(* IEC 61131-3 sources: AXOpen/src/data/ctrl/test, 10 files *)

(* ---- AxoDataCrudTask.st ---- *)
USING AXOpen.Core;
USING AXOpen.Rtc;
USING AxUnit;

NAMESPACE DummyNmspc
        {TestFixture}
        {S7.extern=ReadWrite}
        CLASS DummyClass

            {Test}
            METHOD PUBLIC Create_sets_identifier
                AxUnit.Assert.Equal(TRUE, TRUE);
            END_METHOD

        END_CLASS
END_NAMESPACE

(* ---- AxoDataCrudTaskEntityExistsSatisfiedTests.st ---- *)
USING AXOpen.Core;
USING AXOpen.Data;
USING AxUnit;

NAMESPACE AXOpen.Data
    {TestFixture}
    {S7.extern=ReadWrite}
    CLASS AxoDataCrudTaskEntityExistsSatisfiedTests
        VAR
            _state : AxoDataCrudTaskEntityExistsSatisfied;
        END_VAR

        {Test}
        METHOD PUBLIC Satisfy_sets_status_and_exist_flag
            VAR
                existsAfterFirstRead : BOOL;
                existsAfterSecondRead : BOOL;
            END_VAR

            _state.Satisfy(eAxoTaskState#Done, TRUE);
            existsAfterFirstRead := _state.Exist();
            existsAfterSecondRead := _state.Exist();

            AxUnit.Assert.Equal(eAxoTaskState#Done, _state.Status);
            AxUnit.Assert.Equal(TRUE, existsAfterFirstRead);
            AxUnit.Assert.Equal(FALSE, existsAfterSecondRead);
        END_METHOD

        {Test}
        METHOD PUBLIC Satisfy_with_false_clears_exist_flag
            VAR
                existsAfterRead : BOOL;
            END_VAR

            _state.Satisfy(eAxoTaskState#Busy, FALSE);
            existsAfterRead := _state.Exist();

            AxUnit.Assert.Equal(eAxoTaskState#Busy, _state.Status);
            AxUnit.Assert.Equal(FALSE, existsAfterRead);
            AxUnit.Assert.Equal(FALSE, _state.Exist());
        END_METHOD
    END_CLASS
END_NAMESPACE

(* ---- AxoDataExchangeTaskTests.st ---- *)
USING AXOpen.Core;
USING AXOpen.Rtc;
USING AxUnit;

NAMESPACE AXOpen.Data
    NAMESPACE AxoDataExchangeTaskTests
        {S7.extern=ReadWrite}
        CLASS TestContext IMPLEMENTS IAxoContext
            VAR PROTECTED
                _openCounter : ULINT;
                _closeCounter : ULINT;
                _identityCounter : ULINT;
             END_VAR
            METHOD PUBLIC Open : ULINT
                _openCounter := _openCounter + ULINT#1;
            END_METHOD

            METHOD PUBLIC Close : ULINT
                _closeCounter := _closeCounter + ULINT#1;
            END_METHOD

            METHOD PUBLIC OpenCycleCount : ULINT
                OpenCycleCount := _openCounter;
            END_METHOD

            METHOD PUBLIC ClosedCycleCount : ULINT
                ClosedCycleCount := _closeCounter;
            END_METHOD

            METHOD PUBLIC CreateIdentity : ULINT
                _identityCounter := _identityCounter + ULINT#1;
                CreateIdentity := _identityCounter;
            END_METHOD

            METHOD PUBLIC GetRtc : IAxoRtc ; END_METHOD

            METHOD PUBLIC InjectRtc VAR_INPUT Rtc : IAxoRtc; END_VAR ; END_METHOD

            VAR PRIVATE
                NULL_LOGGER : _NULL_LOGGER;
            END_VAR
            METHOD PUBLIC GetLogger : AXOpen.Logging.IAxoLogger GetLogger := NULL_LOGGER; END_METHOD
            METHOD PUBLIC InjectLogger VAR_INPUT _logger : AXOpen.Logging.IAxoLogger; END_VAR ; END_METHOD
        END_CLASS

        {TestFixture}
        {S7.extern=ReadWrite}
        CLASS AxoDataExchangeTask_Tests
            VAR PROTECTED
                _context : TestContext;
                _dataExchangeTask : AxoDataCrudTask;
            END_VAR

            {Test}
            METHOD PUBLIC InvokeWithIdentifier_sets_identifier
                VAR
                    expected : STRING[254];
                END_VAR
                _dataExchangeTask.Initialize(_context);
                _context.Open();
                expected := 'CreateRecordIdentifier';
                _dataExchangeTask.Invoke(expected);
                _context.Close();
                AxUnit.Assert.Equal(TRUE, _dataExchangeTask.DataEntityIdentifier = expected);
            END_METHOD

        END_CLASS
    END_NAMESPACE
END_NAMESPACE

(* ---- AxoDataExchangeTests.st ---- *)
USING AXOpen.Core;
USING AXOpen.Rtc;
USING AxUnit;

NAMESPACE AXOpen.Data
    NAMESPACE AxoDataExchangeTests
        CLASS TestContext IMPLEMENTS IAxoContext
            VAR PROTECTED
                _openCounter : ULINT;
                _closeCounter : ULINT;
                _identityCounter : ULINT;
             END_VAR
            METHOD PUBLIC Open : ULINT
                _openCounter := _openCounter + ULINT#1;
            END_METHOD

            METHOD PUBLIC Close : ULINT
                _closeCounter := _closeCounter + ULINT#1;
            END_METHOD

            METHOD PUBLIC OpenCycleCount : ULINT
                OpenCycleCount := _openCounter;
            END_METHOD

            METHOD PUBLIC ClosedCycleCount : ULINT
                ClosedCycleCount := _closeCounter;
            END_METHOD

            METHOD PUBLIC CreateIdentity : ULINT
                _identityCounter := _identityCounter + ULINT#1;
                CreateIdentity := _identityCounter;
            END_METHOD

            METHOD PUBLIC GetRtc : IAxoRtc ; END_METHOD

            METHOD PUBLIC InjectRtc VAR_INPUT Rtc : IAxoRtc; END_VAR ; END_METHOD
            VAR PRIVATE
                NULL_LOGGER : _NULL_LOGGER;
            END_VAR
            METHOD PUBLIC GetLogger : AXOpen.Logging.IAxoLogger GetLogger := NULL_LOGGER; END_METHOD
            METHOD PUBLIC InjectLogger VAR_INPUT _logger : AXOpen.Logging.IAxoLogger; END_VAR ; END_METHOD
        END_CLASS

        {TestFixture}
        CLASS AxoDataExchange_Tests
            VAR PROTECTED
                _context : TestContext;
                _dataExchange : AxoDataExchange;
            END_VAR

            {Test}
            METHOD PUBLIC Create_sets_identifier
                VAR
                    expected : STRING[254];
                END_VAR
                _dataExchange.Initialize(_context);
                _context.Open();
                expected := 'CreateRecordIdentifier';
                _dataExchange.Create(expected);
                _context.Close();
                AxUnit.Assert.Equal(_dataExchange.Operation.DataEntityIdentifier, expected);
            END_METHOD

            {Test}
            METHOD PUBLIC Read_sets_identifier
                VAR
                    expected : STRING[254];
                END_VAR
                _dataExchange.Initialize(_context);
                _context.Open();
                expected := 'ReadRecordIdentifier';
                _dataExchange.Read(expected);
                _context.Close();
                AxUnit.Assert.Equal(_dataExchange.Operation.DataEntityIdentifier, expected);
            END_METHOD

            {Test}
            METHOD PUBLIC Update_sets_identifier
                VAR
                    expected : STRING[254];
                END_VAR
                _dataExchange.Initialize(_context);
                _context.Open();
                expected := 'UpdateRecordIdentifier';
                _dataExchange.Update(expected);
                _context.Close();
                AxUnit.Assert.Equal(_dataExchange.Operation.DataEntityIdentifier, expected);
            END_METHOD

            {Test}
            METHOD PUBLIC Delete_sets_identifier
                VAR
                    expected : STRING[254];
                END_VAR
                _dataExchange.Initialize(_context);
                _context.Open();
                expected := 'DeleteRecordIdentifier';
                _dataExchange.Delete(expected);
                _context.Close();
                AxUnit.Assert.Equal(_dataExchange.Operation.DataEntityIdentifier, expected);
            END_METHOD

            {Test}
            METHOD PUBLIC EntityExist_sets_identifier
                VAR
                    expected : STRING[254];
                END_VAR
                _dataExchange.Initialize(_context);
                _context.Open();
                expected := 'EntityExistRecordIdentifier';
                _dataExchange.EntityExist(expected);
                _context.Close();
                AxUnit.Assert.Equal(_dataExchange.Operation.DataEntityIdentifier, expected);
            END_METHOD

            {Test}
            METHOD PUBLIC CreateOrUpdate_sets_identifier
                VAR
                    expected : STRING[254];
                END_VAR
                _dataExchange.Initialize(_context);
                _context.Open();
                expected := 'CreateOrUpdateRecordIdentifier';
                _dataExchange.CreateOrUpdate(expected);
                _context.Close();
                AxUnit.Assert.Equal(_dataExchange.Operation.DataEntityIdentifier, expected);
            END_METHOD
        END_CLASS
    END_NAMESPACE
END_NAMESPACE

(* ---- AxoDataLocalExchangeTest.st ---- *)
USING AXOpen.Messaging.Static;
USING AXOpen.Core;
USING AXOpen.Core.Dummies;
USING AXOpen.Data;

NAMESPACE AXOpen.Data
    CLASS _DataStorage_template EXTENDS AxoDataLocalExchange
        VAR CONSTANT
            LOWBOUND : DINT := 0;
            HIGHBOUND : DINT := 10;
        END_VAR
        VAR PUBLIC
            Payload : _EntityTemplate_;
            Storage : ARRAY[LOWBOUND..HIGHBOUND] OF _EntityTemplate_;
        END_VAR

        METHOD PUBLIC OVERRIDE Create : IAxoTaskState
            VAR_INPUT
                inIdentifier : STRING[254];
            END_VAR
            VAR
                tmpSlot : DINT;
             END_VAR

            dataExchangeTask.Status := eAxoTaskState#Busy;
            operation := eCrudOperation#Create;

            tmpSlot :=THIS.GetFreeSlot();
            IF(tmpSlot >= 0) THEN
                Payload.DataEntityId :=  inIdentifier;
                Storage[tmpSlot] :=  Payload;
                dataExchangeTask.Status := eAxoTaskState#Done;
            ELSE
                dataExchangeTask.Status := eAxoTaskState#Error;
            END_IF;

            Create := dataExchangeTask;
        END_METHOD

        METHOD PUBLIC OVERRIDE Read : IAxoTaskState
            VAR_INPUT
                inIdentifier : STRING[254];
            END_VAR
            VAR
                tmpStorage : REF_TO ARRAY[*] OF IAxoDataEntity;
                tmpEntity : IAxoDataEntity;
                tmpSlot : DINT;
             END_VAR

            dataExchangeTask.Status := eAxoTaskState#Busy;
            operation := eCrudOperation#Read;
            tmpSlot := THIS.LocateSlot(inIdentifier);
            IF(tmpSlot >= LOWBOUND && tmpSlot <= HIGHBOUND) THEN
                Payload := Storage[tmpSlot];
                dataExchangeTask.Status := eAxoTaskState#Done;
            ELSE
                dataExchangeTask.Status := eAxoTaskState#Error;
            END_IF;

            Read := dataExchangeTask;
        END_METHOD

        METHOD PUBLIC OVERRIDE Update : IAxoTaskState
            VAR_INPUT
                inIdentifier : STRING[254];
            END_VAR
            VAR
                tmpSlot : DINT;
            END_VAR
            dataExchangeTask.Status := eAxoTaskState#Busy;
            operation := eCrudOperation#Update;

            tmpSlot := THIS.LocateSlot(inIdentifier);
            IF(tmpSlot >= LOWBOUND && tmpSlot <= HIGHBOUND) THEN
                Payload := Storage[tmpSlot];
                dataExchangeTask.Status := eAxoTaskState#Done;
            ELSE
                dataExchangeTask.Status := eAxoTaskState#Error;
            END_IF;

            Update := dataExchangeTask;
        END_METHOD

        METHOD PUBLIC OVERRIDE Delete : IAxoTaskState
            VAR_INPUT
                inIdentifier : STRING[254];
            END_VAR

            dataExchangeTask.Status := eAxoTaskState#Busy;
            operation := eCrudOperation#Delete;

            Storage[THIS.LocateSlot(inIdentifier)].DataEntityId := '';
            dataExchangeTask.Status := eAxoTaskState#Done;
            Delete := dataExchangeTask;
        END_METHOD

        METHOD PUBLIC OVERRIDE EntityExist : IAxoDataCrudTaskEntityExistState
            VAR_INPUT
                inIdentifier : STRING[254];
            END_VAR
            ;
        END_METHOD

        METHOD PUBLIC OVERRIDE CreateOrUpdate : IAxoTaskState
            VAR_INPUT
                inIdentifier : STRING[254];
            END_VAR
            dataExchangeTask.Status := eAxoTaskState#Done;
            CreateOrUpdate := dataExchangeTask;
        END_METHOD

        METHOD PUBLIC OVERRIDE Restore
            ;
        END_METHOD

        METHOD PRIVATE GetFreeSlot : DINT
            VAR
                i : DINT;
                s : IAxoDataEntity;
            END_VAR
            GetFreeSlot := -1;
            FOR i := LOWBOUND TO HIGHBOUND DO
                IF(Storage[i].DataEntityId = '') THEN
                     GetFreeSlot := i;
                     RETURN;
                END_IF;
            END_FOR;
        END_METHOD

        METHOD PRIVATE LocateSlot : DINT
            VAR_INPUT
                inIdentifier : STRING[254];
            END_VAR
            VAR
                i : DINT;
                s : IAxoDataEntity;
            END_VAR
            LocateSlot := -1;
            FOR i := LOWBOUND TO HIGHBOUND DO
                IF(Storage[i].DataEntityId = inIdentifier) THEN
                    LocateSlot := i;
                     RETURN;
                END_IF;
            END_FOR;
        END_METHOD
    END_CLASS

    {TestFixture}
    {S7.extern=ReadWrite}
    CLASS AxoDataLocalExchangeTests
        VAR
            context : Context;
            rootObject : MockAxoObject;
            storageController : _DataStorage_template;
            s : ARRAY[0..10] OF _EntityTemplate_;
            rtm : MockAxoRtm;
            rtc : MockAxoRtc;
        END_VAR

        {FixtureSetup}
        METHOD PUBLIC TestFixtureSetup
            VAR
                index : INT;
            END_VAR
            context.InitializeRootObject(rootObject);
            context.InjectRtc(rtc);
            context.InjectRtm(rtm);
        END_METHOD

        {Test}
        METHOD PUBLIC create_new_entity_with_identifier
            VAR
                index : INT;
            END_VAR

            storageController.Payload.DataEntityId := 'NON-ID';
            storageController.Payload._hello := 'HEY';
            storageController.Payload._someNumber := 1;
            storageController.Create('ID');

            storageController.Payload.DataEntityId := 'NON-ID';
            storageController.Payload._hello := 'HEY-2';
            storageController.Payload._someNumber := 2;
            storageController.Create('ID-2');

            storageController.Read('ID');

            AxUnit.Assert.Equal(storageController.Payload._hello = 'HEY' , TRUE);
            AxUnit.Assert.Equal(storageController.Payload.DataEntityId = 'ID' , TRUE);
            AxUnit.Assert.Equal(storageController.Payload._someNumber , 1);
        END_METHOD

        {Test}
        METHOD PUBLIC read_new_entity_with_identifier
            VAR
                index : INT;
            END_VAR

            storageController.Payload.DataEntityId := 'NON-ID';
            storageController.Payload._hello := 'HEY';
            storageController.Payload._someNumber := 1;
            storageController.Create('ID');

            storageController.Payload.DataEntityId := 'NON-ID';
            storageController.Payload._hello := 'TO_BE_READ';
            storageController.Payload._someNumber := 2;
            storageController.Create('READ-ID');

            storageController.Read('READ-ID');

            AxUnit.Assert.Equal(storageController.Payload._hello = 'TO_BE_READ' , TRUE);
            AxUnit.Assert.Equal(storageController.Payload.DataEntityId = 'READ-ID' , TRUE);
            AxUnit.Assert.Equal(storageController.Payload._someNumber , 2);
        END_METHOD

        {Test}
        METHOD PUBLIC delet_entity_with_identifier
            VAR
                index : INT;
            END_VAR

            storageController.Payload.DataEntityId := 'NON-ID';
            storageController.Payload._hello := 'HEY';
            storageController.Payload._someNumber := 1;
            storageController.Create('ID');

            storageController.Payload.DataEntityId := 'NON-ID';
            storageController.Payload._hello := 'TO_BE_READ';
            storageController.Payload._someNumber := 2;
            storageController.Create('DELETE-ID');

            storageController.Delete('DELETE-ID');

            storageController.Read('DELETE-ID');

            AxUnit.Assert.Equal( storageController.Read('DELETE-ID').HasError() , TRUE);
        END_METHOD
    END_CLASS

    CLASS _EntityTemplate_ EXTENDS AxoDataEntity
        VAR PUBLIC
            _hello : STRING;
            _someNumber : INT;
        END_VAR
    END_CLASS
    CLASS Context EXTENDS MockAxoContext
        VAR

        END_VAR
        METHOD OVERRIDE Main
            ;
        END_METHOD
    END_CLASS
END_NAMESPACE

(* ---- AxoDataPersistentExchangeTaskTests.st ---- *)
USING AXOpen.Core;
USING AXOpen.Rtc;
USING AxUnit;

NAMESPACE AXOpen.Data
    NAMESPACE AxoDataPersistentExchangeTaskTests
        {S7.extern=ReadWrite}
        CLASS TestContext IMPLEMENTS IAxoContext
            VAR PROTECTED
                _openCounter : ULINT;
                _closeCounter : ULINT;
                _identityCounter : ULINT;
             END_VAR
            METHOD PUBLIC Open : ULINT
                _openCounter := _openCounter + ULINT#1;
            END_METHOD

            METHOD PUBLIC Close : ULINT
                _closeCounter := _closeCounter + ULINT#1;
            END_METHOD

            METHOD PUBLIC OpenCycleCount : ULINT
                OpenCycleCount := _openCounter;
            END_METHOD

            METHOD PUBLIC ClosedCycleCount : ULINT
                ClosedCycleCount := _closeCounter;
            END_METHOD

            METHOD PUBLIC CreateIdentity : ULINT
                _identityCounter := _identityCounter + ULINT#1;
                CreateIdentity := _identityCounter;
            END_METHOD

            METHOD PUBLIC GetRtc : IAxoRtc ; END_METHOD

            METHOD PUBLIC InjectRtc VAR_INPUT Rtc : IAxoRtc; END_VAR ; END_METHOD

            VAR PRIVATE
                NULL_LOGGER : _NULL_LOGGER;
            END_VAR
            METHOD PUBLIC GetLogger : AXOpen.Logging.IAxoLogger GetLogger := NULL_LOGGER; END_METHOD
            METHOD PUBLIC InjectLogger VAR_INPUT _logger : AXOpen.Logging.IAxoLogger; END_VAR ; END_METHOD
        END_CLASS

        {TestFixture}
        {S7.extern=ReadWrite}
        CLASS AxoDataPersistentExchangeTask_Tests
            VAR PROTECTED
                _context : TestContext;
                _dataExchangeTask : AxoDataPersistentCurdTask;
            END_VAR

            {Test}
            METHOD PUBLIC InvokeWithIdentifier_sets_identifier
                VAR
                    expected : STRING[254];
                END_VAR
                _dataExchangeTask.Initialize(_context);
                _context.Open();
                expected := 'UpdateIdentifier';
                _dataExchangeTask.Invoke(expected);
                _context.Close();
                AxUnit.Assert.Equal(TRUE, _dataExchangeTask.DataEntityIdentifier = expected);
            END_METHOD

        END_CLASS
    END_NAMESPACE
END_NAMESPACE

(* ---- AxoDataPersistentExchangeTests.st ---- *)
USING AXOpen.Core;
USING AXOpen.Rtc;
USING AxUnit;

NAMESPACE AXOpen.Data
    NAMESPACE AxoDataPersistentExchangeTests
        {S7.extern=ReadWrite}
        CLASS TestContext EXTENDS Dummies.MockAxoContext
            METHOD PROTECTED OVERRIDE Main
                ;
            END_METHOD
        END_CLASS

        {TestFixture}
        {S7.extern=ReadWrite}
        CLASS AxoDataExchange_Tests
            VAR PROTECTED
                _context : TestContext;
                _rootObject : AxoObject;
                _rtc : AXOpen.Core.Dummies.MockAxoRtc;
                _rtm : AXOpen.Core.Dummies.MockAxoRtm;

                _dataExchange : AxoDataPersistentExchange;

                caller_1 : AxoObject;
                caller_2 : AxoObject;
            END_VAR

            VAR
                _contextBlank : TestContext;
                _dataExchangeBlank : AxoDataPersistentExchange;
                caller_1Blank : AxoObject;
                caller_2Blank : AxoObject;
            END_VAR

            {TestSetup}
            METHOD PUBLIC TestSetup
            // Will be called before MyTest_A AND before Test_B are executed
                _context := _contextBlank;
                _rtm.SetElapsed(LTIME#2s);
                _context.InjectRtm(_rtm);
                _rtc.SetNowUTC(LDATE_AND_TIME#2012-01-12-15:58:12.123);
                _context.InjectRtc(_rtc);
                _context.InitializeRootObject(_rootObject);
                _dataExchange.Run(_rootObject);
                _dataExchange := _dataExchangeBlank;
                caller_1 := caller_1Blank;
                caller_2 := caller_2Blank;
            END_METHOD

            {TestTearDown}
            METHOD PUBLIC TestTearDown
            // Will be called after MyTest_A AND before Test_B where executed
                ;
            END_METHOD

            {FixtureSetup}
            METHOD PUBLIC FixtureSetup
            // Will be called once before the Tests are executed
                ;
            END_METHOD

            {FixtureTearDown}
            METHOD PUBLIC FixtureTearDown
            // Will be called after the Tests where executed
                ;
            END_METHOD

            METHOD PUBLIC RunContextMultipleltipleTimes
                VAR_INPUT
                    cycleCount : INT;
                end_var
                VAR
                    iteration : INT;
                END_VAR
                FOR iteration := 0 TO cycleCount DO
                    _context.Open();
                    _dataExchange.Run(_rootObject);
                    _context.Close();
                END_FOR;
            END_METHOD

            {Test}
            METHOD PUBLIC InvokeRead_NotInvoked_WhenFirstReadDoneNotFinish
                VAR
                    IdentifierCaller_1 : STRING[254];

                    ResultCaller_1 :BOOL;

                    startTime : LDATE_AND_TIME;
                END_VAR
                // initializtion
                startTime := LDATE_AND_TIME#2023-11-11-11:11:11.111;
                _rtc.SetNowUTC(startTime);
                _context.InjectRtc(_rtc);
                caller_1.Run(_rootObject);
                caller_1.Identity :=  _context.CreateIdentity();
                IdentifierCaller_1 := '1';
                _dataExchange.Operation.IsInitialized := true; //simulate intit from .net side

                // needs to simulate + 2 cycles
                THIS.RunContextMultipleltipleTimes(3);

                 //------------------------ INVOKE READ  ------------------------
                _context.Open();
                _dataExchange.Run(_rootObject);

                AxUnit.Assert.Equal(TRUE, _dataExchange.Operation.IsReady());
                ResultCaller_1 := _dataExchange.InvokeRead(caller_1, IdentifierCaller_1);
                AxUnit.Assert.Equal(TRUE, _dataExchange.Operation._EntityId = '');
                AxUnit.Assert.Equal(ResultCaller_1,FALSE);

                _context.Close();

                //------------------------ INVOKE READ  ------------------------
                _context.Open();
                _dataExchange.Run(_rootObject);

                AxUnit.Assert.Equal(TRUE, _dataExchange.Operation.IsReady());
                ResultCaller_1 := _dataExchange.InvokeRead(caller_1, IdentifierCaller_1);
                AxUnit.Assert.Equal(TRUE, _dataExchange.Operation._EntityId = '');
                AxUnit.Assert.Equal(ResultCaller_1,FALSE);

                _context.Close();

                //------------------------ INVOKE READ  ------------------------
                _context.Open();
                _dataExchange.Run(_rootObject);

                AxUnit.Assert.Equal(TRUE, _dataExchange.Operation.IsReady());
                ResultCaller_1 := _dataExchange.InvokeRead(caller_1, IdentifierCaller_1);
                AxUnit.Assert.Equal(TRUE, _dataExchange.Operation._EntityId = '');
                AxUnit.Assert.Equal(ResultCaller_1,FALSE);

                _context.Close();
            END_METHOD

            {Test}
            METHOD PUBLIC InvokeRead_Invoked_WhenFirstReadDoneFinish
                VAR
                    IdentifierCaller_1 : STRING[254];

                    ResultCaller_1 :BOOL;

                    startTime : LDATE_AND_TIME;
                END_VAR
                // initializtion
                startTime := LDATE_AND_TIME#2023-11-11-11:11:11.111;
                _rtc.SetNowUTC(startTime);
                _context.InjectRtc(_rtc);
                caller_1.Run(_rootObject);
                caller_1.Identity :=  _context.CreateIdentity();
                IdentifierCaller_1 := '1';
                _dataExchange.Operation.IsInitialized := true; //simulate intit from .net side

                // needs to simulate + 2 cycles
                THIS.RunContextMultipleltipleTimes(3);

                 //------------------------ INVOKE READ BLOCKED ------------------------
                _context.Open();
                _dataExchange.Run(_rootObject);

                AxUnit.Assert.Equal(TRUE, _dataExchange.Operation.IsReady());
                ResultCaller_1 := _dataExchange.InvokeRead(caller_1, IdentifierCaller_1);
                AxUnit.Assert.Equal(TRUE, _dataExchange.Operation._EntityId = '');
                AxUnit.Assert.Equal(ResultCaller_1,FALSE);

                _context.Close();

                //------------------------ INVOKE READ ENABLED ------------------------

                _dataExchange.SetFirstReadDone(); // firs read done simulation

                _context.Open();
                _dataExchange.Run(_rootObject);

                AxUnit.Assert.Equal(TRUE, _dataExchange.Operation.IsReady());
                ResultCaller_1 := _dataExchange.InvokeRead(caller_1, IdentifierCaller_1); // kicking
                AxUnit.Assert.Equal(TRUE, _dataExchange.Operation._EntityId = IdentifierCaller_1);
                AxUnit.Assert.Equal(ResultCaller_1,FALSE);

                _context.Close();

                //------------------------ INVOKE READ  ------------------------
                _context.Open();
                _dataExchange.Run(_rootObject);

                AxUnit.Assert.Equal(FALSE, _dataExchange.Operation.IsReady());
                ResultCaller_1 := _dataExchange.InvokeRead(caller_1, IdentifierCaller_1); // BUSY => INVOKED
                AxUnit.Assert.Equal(TRUE, _dataExchange.Operation._EntityId = IdentifierCaller_1);
                AxUnit.Assert.Equal(ResultCaller_1,TRUE);

                _context.Close();

            END_METHOD

            {Test}
            METHOD PUBLIC InvokeRead_NotInvoked_CallerHasNoIdentity
                VAR
                    IdentifierCaller_1 : STRING[254];

                    ResultCaller_1 :BOOL;

                    startTime : LDATE_AND_TIME;
                END_VAR
                // initializtion
                startTime := LDATE_AND_TIME#2023-11-11-11:11:11.111;
                _rtc.SetNowUTC(startTime);
                _context.InjectRtc(_rtc);
                caller_1.Run(_rootObject);
                caller_1.Identity := ulint#0;
                IdentifierCaller_1 := '1';
                _dataExchange.Operation.IsInitialized := true; //simulate intit from .net side
                _dataExchange.SetFirstReadDone();

                // needs to simulate + 2 cycles
                THIS.RunContextMultipleltipleTimes(3);

                 //------------------------ INVOKE READ  ------------------------
                _context.Open();
                _dataExchange.Run(_rootObject);

                AxUnit.Assert.Equal(TRUE, _dataExchange.Operation.IsReady());
                ResultCaller_1 := _dataExchange.InvokeRead(caller_1, IdentifierCaller_1);
                AxUnit.Assert.Equal(TRUE, _dataExchange.Operation._EntityId = '');
                AxUnit.Assert.Equal(ResultCaller_1,FALSE);

                _context.Close();

                //------------------------ INVOKE READ  ------------------------
                _context.Open();
                _dataExchange.Run(_rootObject);

                AxUnit.Assert.Equal(TRUE, _dataExchange.Operation.IsReady());
                ResultCaller_1 := _dataExchange.InvokeRead(caller_1, IdentifierCaller_1);
                AxUnit.Assert.Equal(TRUE, _dataExchange.Operation._EntityId = '');
                AxUnit.Assert.Equal(ResultCaller_1,FALSE);

                _context.Close();

                //------------------------ INVOKE READ  ------------------------
                _context.Open();
                _dataExchange.Run(_rootObject);

                AxUnit.Assert.Equal(TRUE, _dataExchange.Operation.IsReady());
                ResultCaller_1 := _dataExchange.InvokeRead(caller_1, IdentifierCaller_1);
                AxUnit.Assert.Equal(TRUE, _dataExchange.Operation._EntityId = '');
                AxUnit.Assert.Equal(ResultCaller_1,FALSE);

                _context.Close();
            END_METHOD

            {Test}
            METHOD PUBLIC InvokeRead_Invoked_CallerHasIdentity
                VAR
                    IdentifierCaller_1 : STRING[254];

                    ResultCaller_1 :BOOL;

                    startTime : LDATE_AND_TIME;
                END_VAR
                // initializtion
                startTime := LDATE_AND_TIME#2023-11-11-11:11:11.111;
                _rtc.SetNowUTC(startTime);
                _context.InjectRtc(_rtc);
                caller_1.Run(_rootObject);
                caller_1.Identity :=  _context.CreateIdentity();
                IdentifierCaller_1 := '1';
                _dataExchange.Operation.IsInitialized := true; //simulate intit from .net side
                _dataExchange.SetFirstReadDone();

                // needs to simulate + 2 cycles
                THIS.RunContextMultipleltipleTimes(3);

                 //------------------------ INVOKE READ  ------------------------
                _context.Open();
                _dataExchange.Run(_rootObject);

                AxUnit.Assert.Equal(TRUE, _dataExchange.Operation.IsReady());
                ResultCaller_1 := _dataExchange.InvokeRead(caller_1, IdentifierCaller_1); // kicking
                AxUnit.Assert.Equal(TRUE, _dataExchange.Operation._EntityId = IdentifierCaller_1);
                AxUnit.Assert.Equal(ResultCaller_1,FALSE);

                _context.Close();

                //------------------------ INVOKE READ  ------------------------
                _context.Open();
                _dataExchange.Run(_rootObject);

                AxUnit.Assert.Equal(FALSE, _dataExchange.Operation.IsReady());
                ResultCaller_1 := _dataExchange.InvokeRead(caller_1, IdentifierCaller_1); // BUSY => INVOKED
                AxUnit.Assert.Equal(TRUE, _dataExchange.Operation._EntityId = IdentifierCaller_1);
                AxUnit.Assert.Equal(ResultCaller_1,TRUE);

                _context.Close();

            END_METHOD

            {Test}
            METHOD PUBLIC ConcurentCall_Update_test
                VAR
                    IdentifierCaller_1 : STRING[254];
                    IdentifierCaller_2 : STRING[254];

                    ResultCaller_1 :BOOL;
                    ResultCaller_2 :BOOL;

                    startTime : LDATE_AND_TIME;
                END_VAR
                // initializtion
                startTime := LDATE_AND_TIME#2023-11-11-11:11:11.111;
                _rtc.SetNowUTC(startTime);
                _context.InjectRtc(_rtc);
                caller_1.Run(_rootObject);
                caller_2.Run(_rootObject);
                caller_1.Identity := _context.CreateIdentity();
                caller_2.Identity := _context.CreateIdentity();
                IdentifierCaller_1 := '1';
                IdentifierCaller_2 := '2';
                _dataExchange.Operation.IsInitialized := true; //simulate intit from .net side
                _dataExchange.SetFirstReadDone();

                // needs to simulate + 2 cycles
                THIS.RunContextMultipleltipleTimes(3);

                 //------------------------ INVOKE READ CONCURRENT ------------------------
                _context.Open();
                _dataExchange.Run(_rootObject);

                AxUnit.Assert.Equal(TRUE, _dataExchange.Operation.IsReady());
                AxUnit.Assert.Equal(FALSE, _dataExchange.Operation.IsBusy());

                ResultCaller_1 := _dataExchange.InvokeUpdate(caller_1, IdentifierCaller_1); // KICKING
                AxUnit.Assert.Equal(FALSE, _dataExchange.Operation.IsReady());
                AxUnit.Assert.Equal(FALSE, _dataExchange.Operation.IsBusy());

                ResultCaller_2 := _dataExchange.InvokeUpdate(caller_2, IdentifierCaller_2); // WAITING

                AxUnit.Assert.Equal(TRUE, _dataExchange.Operation._EntityId = IdentifierCaller_1);
                AxUnit.Assert.Equal(ResultCaller_1,FALSE);
                AxUnit.Assert.Equal(ResultCaller_2,FALSE);

                _context.Close();
                //------------------------ INVOKE SUCCESEED - caller 1. ------------------------
                _context.Open();
                _dataExchange.Run(_rootObject);

                AxUnit.Assert.Equal(FALSE, _dataExchange.Operation.IsReady());
                AxUnit.Assert.Equal(TRUE, _dataExchange.Operation.IsBusy());

                ResultCaller_1 := _dataExchange.InvokeUpdate(caller_1, IdentifierCaller_1); // BUSY - OK
                ResultCaller_2 := _dataExchange.InvokeUpdate(caller_2, IdentifierCaller_2); // WAITING

                AxUnit.Assert.Equal(TRUE, _dataExchange.Operation._EntityId = IdentifierCaller_1);
                AxUnit.Assert.Equal(ResultCaller_1,TRUE);
                AxUnit.Assert.Equal(ResultCaller_2,FALSE);

                _dataExchange.Operation.DoneSignature := _dataExchange.Operation.StartSignature; // remote task done

                _context.Close();
                //------------------------ DONE - caller 1. ------------------------
                _context.Open();
                _dataExchange.Run(_rootObject); // SET DONE STATUS

                AxUnit.Assert.Equal(TRUE, _dataExchange.Operation.IsDone());
                AxUnit.Assert.Equal(FALSE, _dataExchange.Operation.IsReady());

                ResultCaller_1 := _dataExchange.IsUpdateDone(caller_1); // is DONE
                ResultCaller_2 := _dataExchange.InvokeUpdate(caller_2, IdentifierCaller_2); // still WAITING

                AxUnit.Assert.Equal(TRUE, _dataExchange.Operation._EntityId = IdentifierCaller_1);
                AxUnit.Assert.Equal(ResultCaller_1,TRUE);
                AxUnit.Assert.Equal(ResultCaller_2,FALSE);
                _context.Close();
                //------------------------ +1 cycle gap between calls ------------------------
                _context.Open();
                _dataExchange.Run(_rootObject);
                //caller 1 finished not colled any more...
                ResultCaller_2 := _dataExchange.InvokeUpdate(caller_2, IdentifierCaller_2); // still WAITING
                AxUnit.Assert.Equal(FALSE, ResultCaller_2);
                _context.Close();
                //------------------------ +2 cycle gap between calls -----------------------
                _context.Open();
                _dataExchange.Run(_rootObject);
                ResultCaller_2 := _dataExchange.InvokeUpdate(caller_2, IdentifierCaller_2); // still WAITING
                AxUnit.Assert.Equal(FALSE, ResultCaller_2);
                _context.Close();
                //------------------------ Kicking  for caller 2 ------------------------
                _context.Open();
                _dataExchange.Run(_rootObject);
                ResultCaller_2 := _dataExchange.InvokeUpdate(caller_2, IdentifierCaller_2); // Kicking for caller 2
                AxUnit.Assert.Equal(FALSE, ResultCaller_2);

                _context.Close();
                //------------------------ INVOKE SUCCESEED -  caller 2. ------------------------
                _context.Open();
                _dataExchange.Run(_rootObject);
                ResultCaller_1 := _dataExchange.InvokeUpdate(caller_1, IdentifierCaller_1); // will wait
                ResultCaller_2 := _dataExchange.InvokeUpdate(caller_2, IdentifierCaller_2); // invoke success

                AxUnit.Assert.Equal(TRUE, _dataExchange.Operation._EntityId = IdentifierCaller_2);
                AxUnit.Assert.Equal(FALSE, ResultCaller_1);
                AxUnit.Assert.Equal(TRUE, ResultCaller_2);

                _dataExchange.Operation.DoneSignature := _dataExchange.Operation.StartSignature; // remote task done
                _context.Close();
                //------------------------ DONE - caller 2. ------------------------
                _context.Open();
                _dataExchange.Run(_rootObject);
                ResultCaller_1 := _dataExchange.InvokeUpdate(caller_1, IdentifierCaller_1); // will wait
                ResultCaller_2 := _dataExchange.IsUpdateDone(caller_2);

                AxUnit.Assert.Equal(TRUE, _dataExchange.Operation._EntityId = IdentifierCaller_2);
                AxUnit.Assert.Equal(FALSE, ResultCaller_1);
                AxUnit.Assert.Equal(TRUE, ResultCaller_2);

                _context.Close();

            END_METHOD

            {Test}
            METHOD PUBLIC ConcurentCall_Read_test
                VAR
                    IdentifierCaller_1 : STRING[254];
                    IdentifierCaller_2 : STRING[254];

                    ResultCaller_1 :BOOL;
                    ResultCaller_2 :BOOL;

                    startTime : LDATE_AND_TIME;
                END_VAR
                // initializtion
                startTime := LDATE_AND_TIME#2023-11-11-11:11:11.111;
                _rtc.SetNowUTC(startTime);
                _context.InjectRtc(_rtc);
                caller_1.Run(_rootObject);
                caller_2.Run(_rootObject);
                caller_1.Identity := _context.CreateIdentity();
                caller_2.Identity := _context.CreateIdentity();
                IdentifierCaller_1 := '1';
                IdentifierCaller_2 := '2';
                _dataExchange.Operation.IsInitialized := true; //simulate intit from .net side
                _dataExchange.SetFirstReadDone();

                // needs to simulate + 2 cycles
                THIS.RunContextMultipleltipleTimes(3);

                 //------------------------ INVOKE  CONCURRENT ------------------------
                _context.Open();
                _dataExchange.Run(_rootObject);

                AxUnit.Assert.Equal(TRUE, _dataExchange.Operation.IsReady());
                AxUnit.Assert.Equal(FALSE, _dataExchange.Operation.IsBusy());

                ResultCaller_1 := _dataExchange.InvokeRead(caller_1, IdentifierCaller_1); // KICKING
                AxUnit.Assert.Equal(FALSE, _dataExchange.Operation.IsReady());
                AxUnit.Assert.Equal(FALSE, _dataExchange.Operation.IsBusy());

                ResultCaller_2 := _dataExchange.InvokeRead(caller_2, IdentifierCaller_2); // WAITING

                AxUnit.Assert.Equal(TRUE, _dataExchange.Operation._EntityId = IdentifierCaller_1);
                AxUnit.Assert.Equal(ResultCaller_1,FALSE);
                AxUnit.Assert.Equal(ResultCaller_2,FALSE);

                _context.Close();
                //------------------------ INVOKE SUCCESEED - caller 1. ------------------------
                _context.Open();
                _dataExchange.Run(_rootObject);

                AxUnit.Assert.Equal(FALSE, _dataExchange.Operation.IsReady());
                AxUnit.Assert.Equal(TRUE, _dataExchange.Operation.IsBusy());

                ResultCaller_1 := _dataExchange.InvokeRead(caller_1, IdentifierCaller_1); // BUSY - OK
                ResultCaller_2 := _dataExchange.InvokeRead(caller_2, IdentifierCaller_2); // WAITING

                AxUnit.Assert.Equal(TRUE, _dataExchange.Operation._EntityId = IdentifierCaller_1);
                AxUnit.Assert.Equal(ResultCaller_1,TRUE);
                AxUnit.Assert.Equal(ResultCaller_2,FALSE);

                _dataExchange.Operation.DoneSignature := _dataExchange.Operation.StartSignature; // remote task done

                _context.Close();
                //------------------------ DONE - caller 1. ------------------------
                _context.Open();
                _dataExchange.Run(_rootObject); // SET DONE STATUS

                AxUnit.Assert.Equal(TRUE, _dataExchange.Operation.IsDone());
                AxUnit.Assert.Equal(FALSE, _dataExchange.Operation.IsReady());

                ResultCaller_1 := _dataExchange.IsReadDone(caller_1); // is DONE
                ResultCaller_2 := _dataExchange.InvokeRead(caller_2, IdentifierCaller_2); // still WAITING

                AxUnit.Assert.Equal(TRUE, _dataExchange.Operation._EntityId = IdentifierCaller_1);
                AxUnit.Assert.Equal(ResultCaller_1,TRUE);
                AxUnit.Assert.Equal(ResultCaller_2,FALSE);
                _context.Close();
                //------------------------ +1 cycle gap between calls ------------------------
                _context.Open();
                _dataExchange.Run(_rootObject);
                //caller 1 finished not colled any more...
                ResultCaller_2 := _dataExchange.InvokeRead(caller_2, IdentifierCaller_2); // still WAITING
                AxUnit.Assert.Equal(FALSE, ResultCaller_2);
                _context.Close();
                //------------------------ +2 cycle gap between calls -----------------------
                _context.Open();
                _dataExchange.Run(_rootObject);
                ResultCaller_2 := _dataExchange.InvokeRead(caller_2, IdentifierCaller_2); // still WAITING
                AxUnit.Assert.Equal(FALSE, ResultCaller_2);
                _context.Close();
                //------------------------ Kicking read for caller 2 ------------------------
                _context.Open();
                _dataExchange.Run(_rootObject);
                ResultCaller_2 := _dataExchange.InvokeRead(caller_2, IdentifierCaller_2); // Kicking for caller 2
                AxUnit.Assert.Equal(FALSE, ResultCaller_2);

                _context.Close();
                //------------------------ INVOKE SUCCESEED -  caller 2. ------------------------
                _context.Open();
                _dataExchange.Run(_rootObject);
                ResultCaller_1 := _dataExchange.InvokeRead(caller_1, IdentifierCaller_1); // will wait
                ResultCaller_2 := _dataExchange.InvokeRead(caller_2, IdentifierCaller_2); // invoke success

                AxUnit.Assert.Equal(TRUE, _dataExchange.Operation._EntityId = IdentifierCaller_2);
                AxUnit.Assert.Equal(FALSE, ResultCaller_1);
                AxUnit.Assert.Equal(TRUE, ResultCaller_2);

                _dataExchange.Operation.DoneSignature := _dataExchange.Operation.StartSignature; // remote task done
                _context.Close();
                //------------------------ DONE - caller 2. ------------------------
                _context.Open();
                _dataExchange.Run(_rootObject);
                ResultCaller_1 := _dataExchange.InvokeRead(caller_1, IdentifierCaller_1); // will wait
                ResultCaller_2 := _dataExchange.IsReadDone(caller_2);

                AxUnit.Assert.Equal(TRUE, _dataExchange.Operation._EntityId = IdentifierCaller_2);
                AxUnit.Assert.Equal(FALSE, ResultCaller_1);
                AxUnit.Assert.Equal(TRUE, ResultCaller_2);

                _context.Close();

            END_METHOD

        END_CLASS
    END_NAMESPACE
END_NAMESPACE

(* ---- DataExchangeTaskTests.st ---- *)
USING AXOpen.Core;
USING AXOpen.Rtc;
USING AxUnit;

NAMESPACE AXOpen.Data
    NAMESPACE DataExchangeTaskTests
        CLASS TestContext IMPLEMENTS IAxoContext
            VAR PROTECTED
                _openCounter : ULINT;
                _closeCounter : ULINT;
                _identityCounter : ULINT;
             END_VAR
            METHOD PUBLIC Open : ULINT
                _openCounter := _openCounter + ULINT#1;
            END_METHOD

            METHOD PUBLIC Close : ULINT
                _closeCounter := _closeCounter + ULINT#1;
            END_METHOD

            METHOD PUBLIC OpenCycleCount : ULINT
                OpenCycleCount := _openCounter;
            END_METHOD

            METHOD PUBLIC ClosedCycleCount : ULINT
                ClosedCycleCount := _closeCounter;
            END_METHOD

            METHOD PUBLIC CreateIdentity : ULINT
                _identityCounter := _identityCounter + ULINT#1;
                CreateIdentity := _identityCounter;
            END_METHOD

            METHOD PUBLIC GetRtc : IAxoRtc ; END_METHOD

            METHOD PUBLIC InjectRtc VAR_INPUT Rtc : IAxoRtc; END_VAR ; END_METHOD

    METHOD PUBLIC Environment : IAxoContextEnvironment
        ;
    END_METHOD
END_CLASS

        {TestFixture}
        CLASS DataExchangeTask_Tests
            VAR PROTECTED
                _context : TestContext;
                _dataExchangeTask : DataExchangeTask;
            END_VAR

            {Test}
            METHOD PUBLIC InvokeWithIdentifier_sets_identifier
                VAR
                    expected : STRING[254];
                END_VAR
                _dataExchangeTask.Initialize(_context);
                _context.Open();
                expected := 'CreateRecordIdentifier';
                _dataExchangeTask.Invoke(expected);
                _context.Close();
                AxUnit.Assert.Equal(_dataExchangeTask.DataEntityIdentifier, expected);
            END_METHOD

        END_CLASS
    END_NAMESPACE
END_NAMESPACE

(* ---- DataExchangeTests.st ---- *)
USING AXOpen.Core;
USING AXOpen.Rtc;
USING AxUnit;

NAMESPACE ix.framework.data
    NAMESPACE DataExchangeTests
        CLASS TestContext IMPLEMENTS IAxoContext
            VAR PROTECTED
                _openCounter : ULINT;
                _closeCounter : ULINT;
                _identityCounter : ULINT;
             END_VAR
            METHOD PUBLIC Open : ULINT
                _openCounter := _openCounter + ULINT#1;
            END_METHOD

            METHOD PUBLIC Close : ULINT
                _closeCounter := _closeCounter + ULINT#1;
            END_METHOD

            METHOD PUBLIC OpenCycleCount : ULINT
                OpenCycleCount := _openCounter;
            END_METHOD

            METHOD PUBLIC ClosedCycleCount : ULINT
                ClosedCycleCount := _closeCounter;
            END_METHOD

            METHOD PUBLIC CreateIdentity : ULINT
                _identityCounter := _identityCounter + ULINT#1;
                CreateIdentity := _identityCounter;
            END_METHOD

            METHOD PUBLIC GetRtc : IAxoRtc ; END_METHOD

            METHOD PUBLIC InjectRtc VAR_INPUT Rtc : IAxoRtc; END_VAR ; END_METHOD

            METHOD PUBLIC Environment : IAxoContextEnvironment
                ;
            END_METHOD
        END_CLASS

        {TestFixture}
        CLASS DataExchange_Tests
            VAR PROTECTED
                _context : TestContext;
                _dataExchange : DataExchange;
            END_VAR

            {Test}
            METHOD PUBLIC Create_sets_identifier
                VAR
                    expected : STRING[254];
                END_VAR
                _dataExchange.Initialize(_context);
                _context.Open();
                expected := 'CreateRecordIdentifier';
                _dataExchange.Create(expected);
                _context.Close();
                AxUnit.Assert.Equal(_dataExchange.CreateTask.DataEntityIdentifier, expected);
            END_METHOD

            {Test}
            METHOD PUBLIC Read_sets_identifier
                VAR
                    expected : STRING[254];
                END_VAR
                _dataExchange.Initialize(_context);
                _context.Open();
                expected := 'ReadRecordIdentifier';
                _dataExchange.Read(expected);
                _context.Close();
                AxUnit.Assert.Equal(_dataExchange.ReadTask.DataEntityIdentifier, expected);
            END_METHOD

            {Test}
            METHOD PUBLIC Update_sets_identifier
                VAR
                    expected : STRING[254];
                END_VAR
                _dataExchange.Initialize(_context);
                _context.Open();
                expected := 'UpdateRecordIdentifier';
                _dataExchange.Update(expected);
                _context.Close();
                AxUnit.Assert.Equal(_dataExchange.UpdateTask.DataEntityIdentifier, expected);
            END_METHOD

            {Test}
            METHOD PUBLIC Delete_sets_identifier
                VAR
                    expected : STRING[254];
                END_VAR
                _dataExchange.Initialize(_context);
                _context.Open();
                expected := 'DeleteRecordIdentifier';
                _dataExchange.Delete(expected);
                _context.Close();
                AxUnit.Assert.Equal(_dataExchange.DeleteTask.DataEntityIdentifier, expected);
            END_METHOD
        END_CLASS
    END_NAMESPACE
END_NAMESPACE

(* ---- testsomething.st ---- *)
USING AxUnit;
NAMESPACE SomethingRatherThanNothingsTests
    {TestFixture}
    CLASS SomethingTests
    {Test}
    METHOD PUBLIC Testofsomemethod
        ; // AxUnit.Assert.Equal(y, x)
    END_METHOD
END_CLASS
END_NAMESPACE
